# EPICS substitutions: iocBoot/iocRobot/robot.substitutions
file "$(TOP)/db/robot.template"
{
pattern
{  P,        R,      CAMERA_PREFIX,   EXAMPLE_PV_NAME}
{32id:, Robot:,    2bmbSP2:      32id:m1}
}
